KUKA KRL program: GetProcessData.src, GetProcessData.dat

--- GetProcessData.src ---
&ACCESS RVO3
&REL 7
&PARAM DISKPATH = KRC:\R1\Program\CELL\Other
DEF GetProcessData()
   ;FOLD DECL
      DECL INT iProfileID_ABCD
      DECL INT iProfileID_A,iProfileID_B,iProfileID_C,iProfileID_D
      DECL INT iProfileID_AB,iProfileID_AC
      DECL ST_ProcessData stTempData
   ;ENDFOLD (DECL)

   ;FOLD INI

      stTempData = stProcessDataIni

   ;ENDFOLD (INI)

   ;Gdzie deklaracja gstProcessData?

   ;Moim zdaniem te standardowe sygnały i zmienne powinny być zadeklarowane w config.dat
   ;bo w sumie wtedy całkiem do config nie trzeba wchodzić
   ;a zamiast tego GlobalSig.DAT i GlobalVar.DAT

   ;Czy jest sens kodować ID profilu czy lepiej wysyłać osobno kodowane?

   ;Fittings to w sumie jest do całego zamówienia a nie do konkretnego profilu
   ;Dawid i tak będzie wysyłał "FrezujZawias"/"FrezujAut3"
   ;czy jest sens to wysyłać w id profilu czy dla calego zamowienia
   ;Np inLockType #Aut3,#Hook3,#Hook5

   ;Typ klamki nie wiem czy cokolwiek da, bo prawdoodobnie nie jesteSmy w stanie frezowac
   ;tylko 2 wewnetrznych scian w skrzydle. Jest to uniemożliwione przez ustawienie stolu do frezowania
   ;inHandleType lub tylko bit inHandle/inOuterHandle
   ;
   ;

   ;Frame dimensions validation
   IF InRange(inFrameDimX,stRangeFrameDimX) THEN
      stTempData.stFrameDim.rX = inFrameDimX
   ELSE
      HALT ;Invalid process data
   ENDIF
   IF InRange(inFrameDimY,stRangeFrameDimY) THEN
      stTempData.stFrameDim.rY = inFrameDimY
   ELSE
      HALT ;Invalid process data
   ENDIF
   IF InRange(inFrameDimZ,stRangeFrameDimZ,TRUE) THEN
      stTempData.stFrameDim.rZ = inFrameDimZ
   ELSE
      HALT ;Invalid process data
   ENDIF

   ;Leaf dimensions validation
   IF InRange(inLeafDimX,stRangeLeafDimX) THEN
      stTempData.stLeafDim.rX = inLeafDimX
   ELSE
      HALT ;Invalid process data
   ENDIF
   IF InRange(inLeafDimY,stRangeLeafDimY) THEN
      stTempData.stLeafDim.rY = inLeafDimY
   ELSE
      HALT ;Invalid process data
   ENDIF
   IF InRange(inLeafDimZ,stRangeLeafDimZ,TRUE) THEN
      stTempData.stFrameDim.rZ = inLeafDimZ
   ELSE
      HALT ;Invalid process data
   ENDIF

   ;Door side
   SWITCH inDoorSide
      CASE 1
         stTempData.eDoorSide = #Left
      CASE 2
         stTempData.eDoorSide = #Right
      DEFAULT
         HALT ;Invalid process data
   ENDSWITCH

   ;Handle type
   SWITCH inHandleType
      CASE 1
         stTempData.eHandleType = #Pull
      CASE 2
         stTempData.eHandleType = #Lever
      DEFAULT
         HALT ;Invalid process data
   ENDSWITCH

   ;Threshold length
   IF InRange(inThresholdLength,stRangeThresholdLen) THEN
      stTempData.stLeafDim.rX = inLeafDimX
   ELSE
      HALT ;Invalid process data
   ENDIF

   ;ProfileID validation
   IF inProfileID>0 THEN
      stTempData.iProfileID = inProfileID
      iProfileID_ABCD = inProfileID
      iProfileID_A = GetDigit(iProfileID_ABCD,1000)
      iProfileID_B = GetDigit(iProfileID_ABCD,100)
      iProfileID_C = GetDigit(iProfileID_ABCD,10)
      iProfileID_D = GetDigit(iProfileID_ABCD,1)
      iProfileID_AB = iProfileID_A*10 + iProfileID_B
      iProfileID_AC = iProfileID_A*10 + iProfileID_C
   ELSE
      HALT ;Invalid process data
   ENDIF

   ;Type of profile
   SWITCH iProfileID_AB
      CASE 11
         stTempData.eProfileType = #Frame90
      CASE 12
         stTempData.eProfileType = #Frame75
      CASE 21
         stTempData.eProfileType = #Leaf90
      CASE 22
         stTempData.eProfileType = #Leaf75
      CASE 31
         stTempData.eProfileType = #Threshold90
      CASE 32
         stTempData.eProfileType = #Threshold75
      DEFAULT
         HALT ;Invalid process data
   ENDSWITCH

   ;Profile placement
   SWITCH iProfileID_C
      CASE 1
         stTempData.eProfilePlace = #Upper
      CASE 2
         stTempData.eProfilePlace = #Bottom
      CASE 3
         stTempData.eProfilePlace = #Right
      CASE 4
         stTempData.eProfilePlace = #Left
      DEFAULT
         HALT ;Invalid process data
   ENDSWITCH

   ;Type of profile fittings
   SWITCH iProfileID_D
      CASE 1
         stTempData.eProfileFittings = #None
      CASE 2
         stTempData.eProfileFittings = #Hinge
      CASE 3
         stTempData.eProfileFittings = #Aut3
      CASE 4
         stTempData.eProfileFittings = #Hook3
      CASE 5
         stTempData.eProfileFittings = #Hook5
      DEFAULT
         HALT ;Invalid process data
   ENDSWITCH

   ;Profile length
   SWITCH iProfileID_AC
      CASE 11
         ;Frame short profile
         IF InRange(inFrameDimY,stRangeFrameDimY) THEN
            stTempData.rProfileLength = inFrameDimY
         ELSE
            HALT ;Invalid process data
         ENDIF
      CASE 13,14
         ;Frame long profile
         IF InRange(inFrameDimX,stRangeFrameDimX) THEN
            stTempData.rProfileLength = inFrameDimX
         ELSE
            HALT ;Invalid process data
         ENDIF
      CASE 21,22
         ;Leaf short profile
         IF InRange(inLeafDimY,stRangeLeafDimY) THEN
            stTempData.rProfileLength = inLeafDimY
         ELSE
            HALT ;Invalid process data
         ENDIF
      CASE 23,24
         ;Leaf long profile
         IF InRange(inLeafDimX,stRangeLeafDimX) THEN
            stTempData.rProfileLength = inFrameDimX
         ELSE
            HALT ;Invalid process data
         ENDIF
      CASE 32
         ;Threshold profile
         IF InRange(inThresholdLength,stRangeThresholdLen) THEN
            stTempData.rProfileLength = inThresholdLength
         ELSE
            HALT ;Invalid process data
         ENDIF
      DEFAULT
         HALT ;Invalid process data
   ENDSWITCH

   ;Actualize global ProcessData
   gstProcessData = stTempData

END

DEFFCT INT GetDigit(iNumber:IN,iBase:IN)
   ;FOLD DECL
      DECL INT iNumber,iBase,iDigit
      DECL INT iQuotient,iRest
   ;ENDFOLD (DECL)

   ;Example: iNumber=342901 iBase=1000
   ;iRest = 901
   ;iQuotinent = 342
   ;iDigit = 2

   IF iNumber<iBase THEN
      HALT ;Invalid input data
   ENDIF

   ;Get the base quotient
   iRest = Modulo(iNumber,iBase,iQuotient)

   ;Get the base digit
   iDigit = Modulo(iQuotient,10)

   ;Return base digit
   RETURN iDigit

ENDFCT

--- GetProcessData.dat ---
&ACCESS RVO1
&REL 7
&PARAM DISKPATH = KRC:\R1\Program\CELL\Other
DEFDAT  GETPROCESSDATA PUBLIC

;ProcessData structure definition
GLOBAL ENUM E_DoorSide Left,Right
GLOBAL ENUM E_LockType Hook3,Hook5,Aut3
GLOBAL ENUM E_HandleType Lever,Pull
GLOBAL ENUM E_ProfilePlace Left,Right,Upper,Bottom
GLOBAL ENUM E_ProfileFittings None,Hinge,Aut3,Hook3,Hook5
GLOBAL ENUM E_ProfileType Leaf75,Leaf90,Frame75,Frame90,Threshold75,Threshold90
GLOBAL STRUC ST_ProcessData INT iLotNo,ST_Dim3 stFrameDim,stLeafDim,E_DoorSide eDoorSide,E_HandleType eHandleType,REAL rThresholdLength,INT iProfileID,E_ProfileType eProfileType,E_ProfilePlace eProfilePlace,E_ProfileFittings eProfileFittings,REAL rProfileLength

;ProcessData structure declaration
DECL GLOBAL ST_ProcessData gstProcessData={stFrameDim {rX 2100.00,rY 1100.00,rZ 90.0000},stLeafDim {rX 2100.00,rY 1100.00},eDoorSide #Left,eHandleType #Pull,iProfileID 1133,eProfileType #Frame90,eProfilePlace #Right,eProfileFittings #Aut3,rProfileLength 2100.00}

;Init values for ProcessData structure
DECL ST_ProcessData stProcessDataIni={iProfileID -1}

;Frame dimensions ranges
DECL CONST ST_Range stRangeFrameDimX={rMin 1750.00,rMax 2450.00}
DECL CONST ST_Range stRangeFrameDimY={rMin 850.000,rMax 1450.00}
DECL CONST ST_Range stRangeFrameDimZ={rMin 75.0000,rMax 90.0000}

;Leaf dimensions ranges
DECL CONST ST_Range stRangeLeafDimX={rMin 1750.00,rMax 2450.00}
DECL CONST ST_Range stRangeLeafDimY={rMin 850.000,rMax 1450.00}
DECL CONST ST_Range stRangeLeafDimZ={rMin 75.0000,rMax 90.0000}

;Threshold length range
DECL CONST ST_Range stRangeThresholdLen={rMin 760.000,rMax 1030.00}

ENDDAT
